PROGRAM MAIN
VAR
 aTransferLines  : ARRAY[1..3] OF SM_TransferLine;
 
 fbSymbolPathStorage : SymbolPathStorage;
 fbMainStepWorker : FB_StepWorker;
END_VAR

aTransferLines[1](sTLMqttName := 'TL1Synch');
aTransferLines[2](sTLMqttName := 'TL2Synch');
aTransferLines[3](sTLMqttName := 'TL3Synch');

CASE fbMainStepWorker.uiStep OF
	
	eMainWaitStart:
	
		IF Visu.bStartTL1
		THEN
			aTransferLines[1].Execute();
		END_IF
		
		IF Visu.bStartTL2
		THEN
			aTransferLines[2].Execute();
		END_IF
		
		IF Visu.bStartTL3
		THEN
			aTransferLines[3].Execute();
		END_IF
		
		
	
END_CASE

END_PROGRAM

(* stored: Version 1.1.0.1, ProductVersion 3.1.4024.2
   POU MAIN: Id {c83d4c06-b08c-4f63-b878-b3a4e7399e2e}, SpecialFunc None *)
